FUNCTION_BLOCK FB_SampleListener EXTENDS FB_ListenerBase2

VAR
	nMessages: INT;
END_VAR

METHOD OnMessageSent : HRESULT
VAR_INPUT
	fbEvent : REFERENCE TO FB_TcEvent; 
END_VAR
nMessages := nMessages + 1;
END_METHOD

END_FUNCTION_BLOCK

(* stored: Version 1.1.0.1, ProductVersion 3.1.4024.6
   POU FB_SampleListener: Id {43be9d72-438a-4d98-a57c-1dab8a4900a2}, SpecialFunc None
   Method OnMessageSent: Id {1bf4b1ee-e547-4983-aa69-aa4bcbe697c8} *)
